// TIA Portal V19 export
DATA_BLOCK "MES_Manager"   // DB208
// stored: InstanceOfName MES_Manager_FB, InstanceOfType FB
"MES_Manager_FB"
   // VAR
   //    Warning : Struct
   //       Topic1xx_Receive : "MES_Msg_Receive_Topic1xx_Err";
   //       Topic1xx_Send { S7_SetPoint := 'True'} : "MES_Msg_Send_Err";
   //       Topic2xx_Receive : "MES_Msg_Receive_Topic2xx_Err";
   //       Topic2xx_Send { S7_SetPoint := 'True'} : "MES_Msg_Send_Err";
   //       Topic3xx_Receive : "MES_Msg_Receive_Topic3xx_Err";
   //       Topic3xx_Send { S7_SetPoint := 'True'} : "MES_Msg_Send_Err";
   //       Topic4xx_Receive : "MES_Msg_Receive_Topic4xx_Err";
   //       Topic4xx_Send { S7_SetPoint := 'True'} : "MES_Msg_Send_Err";
   //    END_STRUCT;
   //    Lock_Send_Msg_Topic1XX : Bool;
   //    Lock_Send_Msg_Topic2XX : Bool;
   //    Lock_Send_Msg_Topic3XX : Bool;
   //    Lock_Send_Msg_Topic4XX : Bool;
   //    Receive_Msg_Topic1XX { S7_SetPoint := 'True'} : "MES_Receive_Msg_Topic1XX_FB";
   //    Receive_Msg_Topic2XX { S7_SetPoint := 'True'} : "MES_Receive_Msg_Topic2XX_FB";
   //    Receive_Msg_Topic3XX { S7_SetPoint := 'True'} : "MES_Receive_Msg_Topic3XX_FB";
   //    Receive_Msg_Topic4XX { S7_SetPoint := 'True'} : "MES_Receive_Msg_Topic4XX_FB";
   //    Send_Msg_From_Buffer_Topic1XX { S7_SetPoint := 'True'} : "MES_Send_Msg_From_Buffer_FB";
   //    Send_Msg_From_Buffer_Topic2XX { S7_SetPoint := 'True'} : "MES_Send_Msg_From_Buffer_FB";
   //    Send_Msg_From_Buffer_Topic3XX { S7_SetPoint := 'True'} : "MES_Send_Msg_From_Buffer_FB";
   //    Send_Msg_From_Buffer_Topic4XX { S7_SetPoint := 'True'} : "MES_Send_Msg_From_Buffer_FB";
   // END_VAR
BEGIN
END_DATA_BLOCK
